(* Logix 5000 project; controller Chocolate_Packaging_system Emulate 5570 rev 31.11; software revision 31.01 *)

TASK MainTask (continuous, watchdog 500 ms) : MainProgram

MODULES
   Local : Emulate 5570 (ICP 2, rev 31.11)
       : vendor 1 type 0 code 15 (ICP 3, rev 1.1, Output RPI 50 ms)
END_MODULES

VAR_GLOBAL   (* controller tags *)
   Blue_bit : BOOL;
   BLUE_Light : ALIAS FOR Local:3:I.Data[0].3;
   Conveyer_motor : ALIAS FOR Local:3:O.Data[0].0;
   CycleStage : DINT;   // Bring Box =0 Fill Box = 1 Unload Station = 2 Intermediate = 3
   Harshey_bit : BOOL;
   Harshey_hopper : ALIAS FOR Local:3:O.Data[0].1;
   Harshey_trigger : BOOL;
   Level_bit : BOOL;
   LEVEL_SW : ALIAS FOR Local:3:I.Data[0].1;
   Motor_bit : BOOL;
   ons : BOOL;
   ons2 : BOOL;
   ons3 : BOOL;
   ons4 : BOOL;
   Pro_bit : BOOL;
   PRO_SW : ALIAS FOR Local:3:I.Data[0].0;
   Red_bit : BOOL;
   RED_Light : ALIAS FOR Local:3:I.Data[0].2;
   Reeses_bit : BOOL;
   Reeses_hopper : ALIAS FOR Local:3:O.Data[0].2;
   Reeses_trigger : BOOL;
END_VAR

PROGRAM MainProgram   (* main routine MainRoutine *)

ROUTINE CONTROL   (* ladder *)
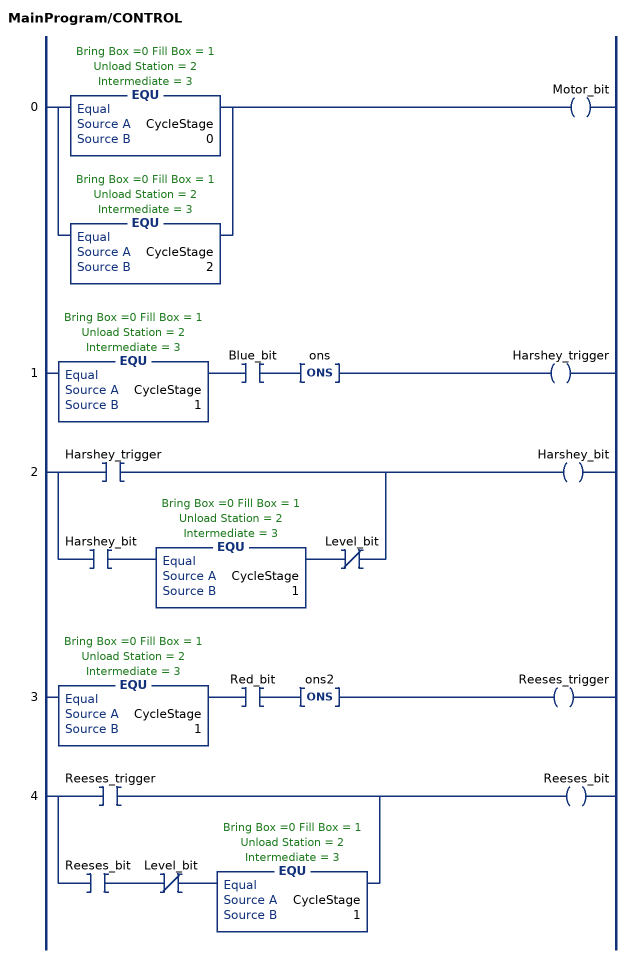
   0: [EQU(CycleStage,0) ,EQU(CycleStage,2) ]OTE(Motor_bit);
   1: EQU(CycleStage,1)XIC(Blue_bit)ONS(ons)OTE(Harshey_trigger);
   2: [XIC(Harshey_trigger) ,XIC(Harshey_bit) EQU(CycleStage,1) XIO(Level_bit) ]OTE(Harshey_bit);
   3: EQU(CycleStage,1)XIC(Red_bit)ONS(ons2)OTE(Reeses_trigger);
   4: [XIC(Reeses_trigger) ,XIC(Reeses_bit) XIO(Level_bit) EQU(CycleStage,1) ]OTE(Reeses_bit);
END_ROUTINE

ROUTINE CYCLE   (* ladder *)
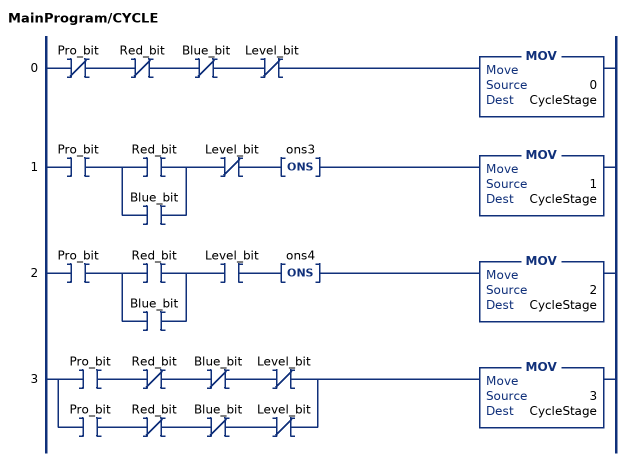
   0: XIO(Pro_bit)XIO(Red_bit)XIO(Blue_bit)XIO(Level_bit)MOV(0,CycleStage);
   1: XIC(Pro_bit)[XIC(Red_bit) ,XIC(Blue_bit) ]XIO(Level_bit)ONS(ons3)MOV(1,CycleStage);
   2: XIC(Pro_bit)[XIC(Red_bit) ,XIC(Blue_bit) ]XIC(Level_bit)ONS(ons4)MOV(2,CycleStage);
   3: [XIC(Pro_bit) XIO(Red_bit) XIO(Blue_bit) XIO(Level_bit) ,XIC(Pro_bit) XIO(Red_bit) XIO(Blue_bit) XIO(Level_bit) ]MOV(3,CycleStage);
END_ROUTINE

ROUTINE IO   (* ladder *)
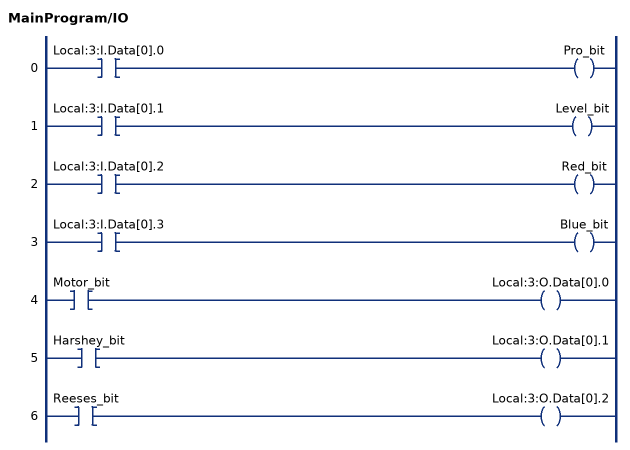
   0: XIC(Local:3:I.Data[0].0)OTE(Pro_bit);
   1: XIC(Local:3:I.Data[0].1)OTE(Level_bit);
   2: XIC(Local:3:I.Data[0].2)OTE(Red_bit);
   3: XIC(Local:3:I.Data[0].3)OTE(Blue_bit);
   4: XIC(Motor_bit)OTE(Local:3:O.Data[0].0);
   5: XIC(Harshey_bit)OTE(Local:3:O.Data[0].1);
   6: XIC(Reeses_bit)OTE(Local:3:O.Data[0].2);
END_ROUTINE

ROUTINE MainRoutine   (* ladder *)
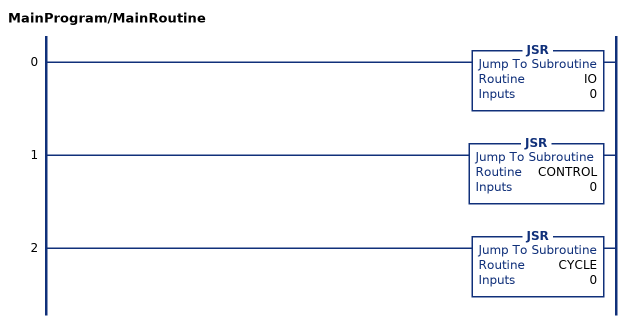
   0: JSR(IO,0);
   1: JSR(CONTROL,0);
   2: JSR(CYCLE,0);
END_ROUTINE
END_PROGRAM
